// TwinCAT 3 PLC project Main
// ProgramVersion: 3.1.4026.10
// libraries:
//   Tc2_EtherCAT, * (Beckhoff Automation GmbH)
//   Tc2_IoFunctions, * (Beckhoff Automation GmbH)
//   Tc2_Math, * (Beckhoff Automation GmbH)
//   Tc2_MC2, * (Beckhoff Automation GmbH)
//   Tc2_NC, * (Beckhoff Automation GmbH)
//   Tc2_Standard, * (Beckhoff Automation GmbH)
//   Tc2_System, * (Beckhoff Automation GmbH)
//   Tc2_Utilities, * (Beckhoff Automation GmbH)
//   Tc3_EventLogger, * (Beckhoff Automation GmbH)
//   Tc3_McCollisionAvoidance, * (Beckhoff Automation GmbH)
//   Tc3_McCoordinatedMotion, * (Beckhoff Automation GmbH)
//   Tc3_Module, * (Beckhoff Automation GmbH)
//   Tc3_XTS_Utility, * (Beckhoff Automation GmbH)
// project tree:
//   DUTs/delete/ MainCommands_typ.TcDUT (not stored), MainStateMachine_enum.TcDUT, MainState_enum.TcDUT (not stored), MediatorGroupStatus.TcDUT (not stored), MotionParameters_typ.TcDUT (not stored), MoverCommandType_enum.TcDUT (not stored), MoverState_enum.TcDUT (not stored), PositionTriggerStats_typ.TcDUT (not stored), StationStats_typ.TcDUT (not stored), TrackCyclicState.TcDUT (not stored), TrackInfo.TcDUT (not stored), TrackState.TcDUT (not stored), UserStationsMonitor.TcDUT
//   DUTs/ M1Detection.TcDUT, MoverControlFlags.TcDUT, MoverSequence.TcDUT (not stored), StationSequence.TcDUT, XTSSequence.TcTLEO
//   / GlobalTextList.TcGTLO (not stored), PlcTask.TcTTO (not stored)
//   GVLs/ GVL.TcGVL, HMI.TcGVL, IOGVL.TcGVL, PersistentGVL.TcGVL, SafetyGVL.TcGVL
//   ITFs/ iMoverList.TcIO, iMover.TcIO (not stored), iTrack.TcIO
//   POUs/ Main.TcPOU
//   POUs/XTS/ Mover.TcPOU, Station.TcPOU

// ---- DUTs/delete/MainStateMachine_enum.TcDUT
{attribute 'strict'}
{attribute 'to_string'}
TYPE MainStateMachine_enum :
(
	MS_DISABLED			:= 0,
	MS_INITIALIZING		:= 10,
	MS_ENABLED			:= 20,
	MS_RUN				:= 30,
	MS_STOPPING			:= 40,
	MS_STOPPED			:= 50,
	MS_DISABLING		:= 60,
	MS_ERROR			:= 70,
	MS_DEBUG			:= 80	
);
END_TYPE

// ---- DUTs/delete/UserStationsMonitor.TcDUT
TYPE UserStationsMonitor :
STRUCT
	
bmoverAtStation		: ARRAY[0..GVL.NUM_STATIONS] OF BOOL;
nmoverAtStation		: ARRAY[0..GVL.NUM_STATIONS] OF UDINT;


END_STRUCT
END_TYPE

// ---- DUTs/M1Detection.TcDUT
{attribute 'qualified_only'}
{attribute 'strict'}
{attribute 'to_string'}
TYPE M1Detection :
(
	Read,
	ReadBuffer,
	Analyze,
	Write,
	WriteBuffer,
	Done,
	Error
	
);
END_TYPE

// ---- DUTs/MoverControlFlags.TcDUT
TYPE MoverControlFlags :
STRUCT

	loadTray_Busy		: BOOL;			// To the machine to check Sensor
	loadTray_Complete	: BOOL;			// From Sensor is TRUE
	inspectTray_Busy	: BOOL;			// Read the state of the sensor TRUE/FALSE
	inspectTray_Complate: BOOL;			// From Camera that tray is done being measured
	loadArea1_Busy		: BOOL;			// TO Robot 1 to start working
	loadArea1_Complete	: BOOL;			// FROM Robot 1 that placing parts has completed
	loadArea2_Busy		: BOOL;			// TO Robot 2 to start working
	loadArea2_Complete	: BOOL;			// FROM Robot 1 that placing parts has completed
	loadArea3_Busy		: BOOL;			// TO Robot 3 to start working
	loadArea3_Complete	: BOOL;			// FROM Robot 1 that placing parts has completed
	loadArea4_Busy		: BOOL;			// TO Robot 4 to start working
	loadArea4_Complete	: BOOL;			// From Robot 1 that placing parts has completed
	unloadTray_Busy		: BOOL;			// To Robot 5 to start working
	unloadTray_Complete	: BOOL;			// From Robot 5. Tray is unloaded



END_STRUCT
END_TYPE

// ---- DUTs/StationSequence.TcDUT
{attribute 'qualified_only'}
{attribute 'strict'}
TYPE StationSequence :
(
	Idle,
	MoverPresent,
	RobotActive,
	DischargeMover,
	Error		
);
END_TYPE

// ---- DUTs/XTSSequence.TcTLEO
{attribute 'qualified_only'}
{attribute 'strict'}
{attribute 'to_string'}
TYPE XTSSequence :
(
	Off,
	EnableMovers,
	EnableGroup,
	AddAxes,
	RemoveAxes,
	RemovedAxes,
	DisableMovers,
	Disabled,
	Start,
	Run,
	Stop,
	Stopping,
	Paused,
	Standby,
	Error,
	Waiting
);
END_TYPE

// ---- GVLs/GVL.TcGVL
{attribute 'qualified_only'}
VAR_GLOBAL CONSTANT
	pXtsProcessingUnit 			: OTCID	:= 16#01010020;	 
	TRACK_LENGTH 				: LREAL := 7000; // This should be set to the exact length [mm] of the track system
	NUM_MOVERS   				: USINT := 20;   // This should be set to the exact number of movers on the system
	
	// The following should be set to a value **equal to or greater than** the number of objectives needed
	NUM_POSITIONTRIGGERS		: USINT := 10;	// Position Triggers
	NUM_STATIONS				: USINT := 8;	// Stations
	NUM_ZONES					: USINT := 10;	// Zones

	// Station constants
	startStation				: USINT	:= 1;		// set this number to the index of the station all movers should start from
	stationTolerance			: LREAL	:= 1;		// set to number of millimeters tolerance for mover at station
	zeroSpeed					: LREAL	:= 10.0;	// tolerance for definition of not moving
END_VAR

VAR_GLOBAL
	Mover					: ARRAY[1..GVL.NUM_MOVERS] OF Mover;
	Station					: ARRAY[1..GVL.NUM_STATIONS] OF station;
	dsMoverControlFlags		: MoverControlFlags;
END_VAR

// ---- GVLs/HMI.TcGVL
{attribute 'qualified_only'}
VAR_GLOBAL
	Start					: BOOL;
	ReStart					: BOOL;
	Stop					: BOOL;
	Resume					: BOOL;
	ResetXTS_Error			: BOOL;
	dsMoverControlFlags		: MoverControlFlags;
	ShuttleMover			: BOOL;
	MachineState			: STRING;
	AutoMode				: BOOL;
	
	//Linked to SAFETY Alias
	LockDoors		AT %Q*	: BOOL;		
	
END_VAR

// ---- GVLs/IOGVL.TcGVL
{attribute 'qualified_only'}
VAR_GLOBAL
	
//INPUTS
iTrayDetectSensor	AT %I*	:	BOOL;
iDoor1Opened		AT %I*	:	BOOL;		
iDoor2Opened		AT %I*	:	BOOL;
iDoor3Opened		AT %I*	:	BOOL;
iDoor4Opened		AT %I*	:	BOOL;
iMainAirPressure 	AT %I*	:	BOOL;

//------XTS Power Monitor Breakers	
//- EL1809 Mod1
iCircuitBreaker24VDC			AT %I*	:	BOOL;
iCircuitBreakerSafety			AT %I*	:	BOOL;
iXTS_Module1					AT %I*	:	BOOL;
iXTS_Module2					AT %I*	:	BOOL;
iXTS_Module3					AT %I*	:	BOOL;
iXTS_Module4					AT %I*	:	BOOL;
iXTS_Module5					AT %I*	:	BOOL;
iXTS_Module6					AT %I*	:	BOOL;
iLubricationOn					AT %I*	:	BOOL;
//- EL1809 Mod2
iPowerSupply48VDC1				AT %I*	:	BOOL;
iPowerSupply48VDC2				AT %I*	:	BOOL;
iPowerSupply48VDC3				AT %I*	:	BOOL;
iLubricationLevelOK				AT %I*	:	BOOL;
iLubricationDone				AT %I*	:	BOOL;
iCircuitBreaker48VDC1			AT %I*	:	BOOL;
iCircuitBreaker48VDC2			AT %I*	:	BOOL;
iCircuitBreaker48VDC3			AT %I*	:	BOOL;
iCircuitBreakerXTSModule1		AT %I*	:	BOOL;
iCircuitBreakerXTSModule2		AT %I*	:	BOOL;
iCircuitBreakerXTSModule3		AT %I*	:	BOOL;
iCircuitBreakerXTSModule4		AT %I*	:	BOOL;
iCircuitBreakerXTSModule5		AT %I*	:	BOOL;
iCircuitBreakerXTSModule6		AT %I*	:	BOOL;
iBrakeResistorON				AT %I*	:	BOOL;

//-----------------------------------------------------------------------------------------------------------------------------------
//OUTPUTS
oBacklight1			AT %Q*	:	BOOL;
oBacklight2			AT %Q*	:	BOOL;
oBacklight3			AT %Q*	:	BOOL;
oBacklight4			AT %Q*	:	BOOL;
oBacklight5			AT %Q*	:	BOOL;
oBacklight6			AT %Q*	:	BOOL;
oBacklight7			AT %Q*	:	BOOL;
oBacklight8			AT %Q*	:	BOOL;
oBacklight9			AT %Q*	:	BOOL;
oBacklight10		AT %Q*	:	BOOL;
oBacklight11		AT %Q*	:	BOOL;
oBacklight12		AT %Q*	:	BOOL;
oBacklight13		AT %Q*	:	BOOL;
oBacklight14		AT %Q*	:	BOOL;
oBacklight15		AT %Q*	:	BOOL;
oBacklight16		AT %Q*	:	BOOL;
oEStopLight			AT %Q*	:	BOOL;
oConveyor			AT %Q*	:	BOOL;
oLubeON				AT %Q*	:	BOOL;

END_VAR

// ---- GVLs/PersistentGVL.TcGVL
{attribute 'qualified_only'}

VAR_GLOBAL RETAIN
	
TimesAroundTrackCounter		: INT;

END_VAR

// ---- GVLs/SafetyGVL.TcGVL
{attribute 'qualified_only'}
VAR_GLOBAL
	
//OUTPUTS TO SAFETY GROUP
err_ack			AT %Q*	:	BOOL;
run				AT %Q*	:	BOOL := TRUE;
DoorsClosed 	AT %Q*	:	BOOL;
ResetCurtains	AT %Q*	:	BOOL;

//INPUTS FROM SAFETY GROUP
CurtainsOK		AT %I*	:	BOOL;
AllSafetyOK		AT %I*	:	BOOL;
EStopStatus		AT %I*	:	BOOL;
DoorsLocked		AT %I*	:	BOOL;

END_VAR

// ---- ITFs/iMoverList.TcIO
INTERFACE iMoverList

METHOD ActivateAllTrack : BOOL
VAR_INPUT
	Track	: REFERENCE TO Track;
END_VAR
END_METHOD

METHOD ApplyAllParameterSet : iMoverList
VAR_INPUT
	ParameterSet		: MotionParameters_typ;
END_VAR
END_METHOD

METHOD Contains : BOOL
VAR_INPUT
	
	Mover		: REFERENCE TO delete_Mover;

END_VAR
END_METHOD

METHOD DestinationStation : iMoverList
VAR_INPUT
	Destination	: REFERENCE TO delete_Station;
END_VAR
END_METHOD

METHOD DisableAll : iMoverList
END_METHOD

METHOD EnableAll : iMoverList
END_METHOD

METHOD GetMoverByLocation : REFERENCE to delete_Mover
VAR_INPUT
    Index     : USINT;                // 0 is find the first closest mover, 1 is find the second closest mover, 2 is find the third, etc. etc. etc.
    Position  : LREAL;                // Fixed track position from which to search for movers by proximity
    Direction : Tc2_MC2.MC_Direction; // Positive = find the most positive mover whose position is less than the Input. Negative = find the most negative mover whose position is greater than the input
END_VAR
END_METHOD

METHOD HaltAll : iMoverList
END_METHOD

PROPERTY IsAllMoversDisabled : bool
GET
END_GET
END_PROPERTY

PROPERTY IsAllMoversHalted : bool
GET
END_GET
END_PROPERTY

PROPERTY IsAllMoversReady : BOOL
GET
END_GET
END_PROPERTY

PROPERTY IsAllTrackReady : BOOL
GET
END_GET
END_PROPERTY

METHOD LogicalComplement : MoverList
VAR_INPUT
END_VAR
END_METHOD

METHOD LogicalDifference : MoverList
VAR_INPUT
	
	MoverList		: MoverList;

END_VAR
END_METHOD

METHOD LogicalIntersect : MoverList
VAR_INPUT
	
	MoverList		: MoverList;

END_VAR
END_METHOD

METHOD LogicalUnion : MoverList
VAR_INPUT
	
	MoverList		: MoverList;

END_VAR
END_METHOD

METHOD MoveAllToPosition : iMoverList
VAR_INPUT

    DestinationPosition : LREAL; // position on track for all shuttles to move towards	

END_VAR
END_METHOD

METHOD MoveAllToStation : iMoverList
VAR_INPUT

    DestinationStation : REFERENCE TO delete_Station;

END_VAR
END_METHOD

METHOD MoveAllVelocity : iMoverList
VAR_INPUT

    Velocity : LREAL;

END_VAR
END_METHOD

METHOD SetAllAcceleration : iMoverList
VAR_INPUT

    Acceleration : LREAL;

END_VAR
END_METHOD

METHOD SetAllDeceleration : iMoverList
VAR_INPUT

    Deceleration : LREAL;

END_VAR
END_METHOD

METHOD SetAllDirection : iMoverList
VAR_INPUT

    Direction : Tc3_Mc3Definitions.MC_DIRECTION;

END_VAR
END_METHOD

METHOD SetAllGap : iMoverList
VAR_INPUT
	Gap : LREAL;
END_VAR
END_METHOD

METHOD SetAllGapMode : iMoverList
VAR_INPUT
    Mode	: MC_GAP_CONTROL_MODE;
END_VAR
END_METHOD

METHOD SetAllJerk : iMoverList
VAR_INPUT

    Jerk : LREAL;

END_VAR
END_METHOD

METHOD SetAllVelocity : iMoverList
VAR_INPUT

    Velocity : LREAL;

END_VAR
END_METHOD

{attribute 'monitoring' := 'call'}
PROPERTY TrackedMoverCount : USINT
GET
END_GET
END_PROPERTY

PROPERTY TrackedMovers : ARRAY[0..GVL.NUM_MOVERS - 1] OF POINTER TO delete_Mover
GET
END_GET
END_PROPERTY

METHOD UnregisterAll : BOOL
VAR_INPUT
END_VAR
END_METHOD

END_INTERFACE

// ---- ITFs/iTrack.TcIO
INTERFACE iTrack

PROPERTY CurrentMoverCount : DINT
GET
END_GET
END_PROPERTY

PROPERTY CurrentMoverList : iMoverList
GET
END_GET
END_PROPERTY

METHOD Cyclic : BOOL
VAR_INPUT
END_VAR
END_METHOD

PROPERTY Id : INT
GET
END_GET
SET
END_SET
END_PROPERTY

PROPERTY isInitialized : bool
GET
END_GET
END_PROPERTY

PROPERTY OTCID : OTCID
GET
END_GET
SET
END_SET
END_PROPERTY

METHOD RegisterMover : BOOL
VAR_INPUT
    NewMover : REFERENCE TO delete_Mover;
END_VAR
VAR
END_VAR
END_METHOD

METHOD UnregisterAll : BOOL
VAR_INPUT
END_VAR
END_METHOD

METHOD UnregisterMover : BOOL
VAR_INPUT
    RemovingMover : REFERENCE TO delete_Mover;
END_VAR
VAR
END_VAR
END_METHOD

END_INTERFACE

// ---- POUs/XTS/Station.TcPOU
FUNCTION_BLOCK Station
VAR_INPUT
	Position		: LREAL;
	bMoveToNext		: BOOL;
	bMoveToStart	: BOOL;
	bMoveToQueue	: BOOL;
END_VAR
VAR_OUTPUT
	CurrentMover	: UDINT;
END_VAR
VAR
	Step			: StationSequence;
	i				: USINT;
	PosLow			: LREAL;
	PosHigh			: LREAL;
END_VAR

(* this function block handles each station *)

PosLow		:= Position - ( GVL.stationTolerance / 2 );
IF PosLow < 0 THEN
	PosLow	:= GVL.TRACK_LENGTH + PosLow;
END_IF
PosHigh		:= Position + ( GVL.stationTolerance / 2 );


CASE Step OF 
//-----------------------------------------------------------------------------------------------------------------------	
	StationSequence.Idle:
		// loop through all movers checking position
		FOR i := 1 TO GVL.NUM_MOVERS DO
			IF GVL.Mover[i].Ready
			AND ( GVL.Mover[i].Step = MoverSequence.AtStart OR GVL.Mover[i].Step = MoverSequence.AtStation )
			AND ABS(GVL.Mover[i].Velocity) < GVL.zeroSpeed THEN
				IF PosLow < PosHigh THEN
					IF GVL.Mover[i].Position > PosLow
					AND GVL.Mover[i].Position < PosHigh THEN
						CurrentMover	:= i;
						Step			:= StationSequence.MoverPresent;
					END_IF
				ELSE
					// station position is close to rollover
					IF GVL.Mover[i].Position > PosLow
					OR GVL.Mover[i].Position < PosHigh THEN
						CurrentMover	:= i;
						Step			:= StationSequence.MoverPresent;
					END_IF
				END_IF
			END_IF
		END_FOR
		
//-----------------------------------------------------------------------------------------------------------------------	
	StationSequence.MoverPresent:
		// robot tasks complete, discharge mover
		IF bMoveToNext THEN									
			Step	:= StationSequence.Idle;
			bMoveToNext := FALSE;
			GVL.Mover[CurrentMover].toNext	:= TRUE;		// request mover move to next station
		END_IF
		
		IF bMoveToStart THEN
			Step	:= StationSequence.Idle;
			bMoveToStart := FALSE;
			GVL.Mover[CurrentMover].toStart	:= TRUE;		// request mover move to Start station
		END_IF
		
		IF bMoveToQueue THEN
			Step	:= StationSequence.Idle;
			bMoveToQueue := FALSE;
			GVL.Mover[CurrentMover].toQueue	:= TRUE;
		END_IF

		
//-----------------------------------------------------------------------------------------------------------------------		
	StationSequence.DischargeMover:
		// request mover move to next station
		//GVL.Mover[CurrentMover].toNext	:= TRUE;
		// verify mover has left
		IF GVL.Mover[CurrentMover].Busy
			AND GVL.Mover[CurrentMover].Position > (Position + GVL.stationTolerance / 2)
			AND GVL.Mover[CurrentMover].Velocity > GVL.zeroSpeed THEN
			Step	:= StationSequence.Idle;
		END_IF
		
END_CASE

END_FUNCTION_BLOCK

// ---- POUs/XTS/Mover.TcPOU
FUNCTION_BLOCK Mover
VAR_INPUT
	Enable			: BOOL;				// Request mover enable
	toStart			: BOOL;				// Request mover go to start position
	toNext			: BOOL;				// Request mover go to next station	
	toStop			: BOOL;				// Request mover to stop - meaning the movers will be stop, removed from group, and power will be shutdown to the track via an E-Stop or HMI.Stop	
	toPause			: BOOL;				// Request mover to pause	
	toDisable		: BOOL;				// Request mover to disable power	
	toQueue			: BOOL;				// Request current mover at starting station to join the back of the queue
	toReset			: BOOL;				// Request current mover at starting station to join the back of the queue
	toIncreaseSpeed	: BOOL;
END_VAR
VAR_OUTPUT
	Enabled			: BOOL;				// Mover confirmed enabled
	Ready			: BOOL;				// Mover is enabled and ready to accept motion commands
	Busy			: BOOL;				// Mover is processing a command or changing state
	Position		: LREAL;			// Current mover position
	Velocity		: LREAL;			// Current mover velocity                                	
	Error			: UDINT;			// errorID of the active error
	Step			: MoverSequence;	// Mover's step within sequence                                	
	AxisReference	: AXIS_REF;			// Motion link variable. Left as output so the link can be made directly, and accessed by external code
	TargetStation	: USINT;
END_VAR
VAR
	// Motion commands
	fbPower					: MC_Power;
	fbReset					: MC_Reset;
	fbHaltCA				: MC_HaltCA;
	fbMoveAbsCA				: MC_MoveAbsoluteCA;
	fbMoveAbsCABlended		: MC_MoveAbsoluteCA;
	fbMoveAbsCABlended2		: MC_MoveAbsoluteCA;
	
	MoveCommandVel			: LREAL := 1000;
	PosLow					: LREAL;
	PosHigh					: LREAL;
	bDummySpeedTest			: BOOL;
	
END_VAR

(* this function block handles each Mover's axis *)

	AxisReference.ReadStatus();
	Enabled		:= NOT AxisReference.Status.Disabled;
	Ready		:= AxisReference.Status.NotMoving AND NOT AxisReference.Status.Error AND NOT AxisReference.Status.Disabled;
	Busy		:= AxisReference.Status.Moving;
	Position	:= AxisReference.NcToPlc.ModuloActPos;
	Velocity	:= AxisReference.NcToPlc.ActVelo;
	Error		:= AxisReference.NcToPlc.ErrorCode;
	
	IF Step = MoverSequence.AtStart AND toQueue THEN
		Step := MoverSequence.MovingToQueue;
		toQueue := FALSE;
	END_IF
	
	IF toStop OR toPause THEN
		fbMoveAbsCA.Execute			:= FALSE;
		fbMoveAbsCABlended.Execute	:= FALSE;
		fbHaltCA.Execute 			:= TRUE;
		fbHaltCA.Deceleration 		:= 1E4;
		IF toStop THEN
			Step := MoverSequence.Stopping;
		ELSIF toPause THEN
			Step := MoverSequence.Pausing;
		END_IF
	END_IF
	
	IF toReset THEN
		Step := MoverSequence.Reset;
		toReset := FALSE;
	END_IF
	

CASE Step OF
//-----------------------------------------------------------------------------------------------------------------------
	MoverSequence.Reset:	
	
		fbReset.Execute := TRUE;
		IF fbReset.Busy THEN
			Step := MoverSequence.Resetting;
		END_IF
	
//---------------------------------
	MoverSequence.Resetting:	
	
	IF fbReset.Done THEN
		fbReset.Execute := FALSE;
		Step := MoverSequence.Waiting;
	END_IF

//-----------------------------------------------------------------------------------------------------------------------
	MoverSequence.MovingToQueue:	
	
		IF NOT fbMoveAbsCA.Busy AND NOT fbMoveAbsCA.Done THEN			//Add additional condition that the doors are not unlcoked
			fbMoveAbsCA.Execute			:= TRUE;
			fbMoveAbsCA.Position		:= GVL.Station[GVL.startStation].Position+2000;
			fbMoveAbsCA.Velocity		:= MoveCommandVel;										// parameterize
			fbMoveAbsCA.Direction		:= MC_Positive_Direction;						// usually positive
		END_IF
			// check for error
		IF fbMoveAbsCA.Error THEN
			Error				:= fbMoveAbsCA.ErrorId;
			Step				:= MoverSequence.Error;
			fbMoveAbsCA.Execute	:= FALSE;
		END_IF
		// check for move complete THEN proceed to starting station
		IF fbMoveAbsCA.Busy AND Position > 1500.0 AND Position < 6900.0 THEN 		//When mover sits at position 0 the values jump +-0 so an asdditional condition must be used
			fbMoveAbsCABlended.Execute		:= TRUE;
			fbMoveAbsCABlended.Position		:= GVL.Station[GVL.startStation].Position;
			fbMoveAbsCABlended.Velocity		:= MoveCommandVel;
			fbMoveAbsCABlended.BufferMode	:= mcAborting;
			fbMoveAbsCABlended.Direction 	:= MC_Positive_Direction;
			Step							:= MoverSequence.AtQueue;
		END_IF
		
//---------------------------------
	MoverSequence.AtQueue:	
	
		IF fbMoveAbsCABlended.Busy THEN
			fbMoveAbsCABlended.Execute			:= FALSE;
			fbMoveAbsCA.Execute					:= FALSE;
			Step								:= MoverSequence.MovingToStart;
		END_IF
	
//-----------------------------------------------------------------------------------------------------------------------
	MoverSequence.Stopping:	
		//RESULT OF PRESSING ESTOP
		IF fbHaltCA.Done OR AxisReference.Status.StandStill OR AxisReference.Status.NotMoving THEN
			fbHaltCA.Execute 	:= FALSE;
			toStart				:= FALSE;
			toNext				:= FALSE;
			toStop				:= FALSE;
			Step := MoverSequence.Disabling;
		END_IF
			
//---------------------------------
	MoverSequence.Disabling:		
	 	//RESULT OF PRESSING ESTOP
		IF toDisable THEN
			Enable						:= FALSE;
			fbPower.Enable				:= FALSE;
			fbPower.Enable_Positive		:= FALSE;
			fbPower.Enable_Negative		:= FALSE;
			fbPower.BufferMode			:= MC_Aborting;
			fbPower.Override			:= 100;
			IF AxisReference.Status.Disabled THEN
				toDisable := FALSE;
				Step := MoverSequence.Off;
			END_IF
		END_IF
			
//-----------------------------------------------------------------------------------------------------------------------
	MoverSequence.Pausing:	
	
		IF fbHaltCA.Done THEN
			fbHaltCA.Execute 	:= FALSE;
			toStart				:= FALSE;
			toNext				:= FALSE;
			toPause				:= FALSE;
			Step := MoverSequence.OFF;
		END_IF

//---------------------------------
	MoverSequence.Off:
		// when enable request is true, use MC_Power function block
		IF Enable THEN
			fbPower.Enable_Positive := TRUE;
			fbPower.Enable := TRUE;
		END_IF
		IF Enabled THEN
			Step	:= MoverSequence.Idle;
		END_IF
		
//---------------------------------	
	MoverSequence.Idle:
		// ready and awaiting either toStart or toNext
		IF toStart THEN
			TargetStation		:= GVL.startStation;
			Step				:= MoverSequence.MovingToStart;
		ELSIF toNext THEN
			Step				:= MoverSequence.MovingToStation;
		END_IF
		
//-----------------------------------------------------------------------------------------------------------------------	
	MoverSequence.MovingToStart:
		// move absolute with collision avoidance to start station
		IF NOT fbMoveAbsCA.Busy AND NOT fbMoveAbsCA.Done THEN	
			fbMoveAbsCA.Execute		:= TRUE;
			fbMoveAbsCA.Position	:= GVL.Station[GVL.startStation].Position;
			fbMoveAbsCA.Velocity	:= MoveCommandVel;							// parameterize
			fbMoveAbsCA.Direction	:= MC_Positive_Direction;		// usually positive
		END_IF
		// check for error
		IF fbMoveAbsCA.Error THEN
			Error				:= fbMoveAbsCA.ErrorId;
			Step				:= MoverSequence.Error;
			fbMoveAbsCA.Execute	:= FALSE;
		END_IF
		IF fbMoveAbsCA.Busy AND Position > GVL.Station[8].Position OR Position < GVL.Station[1].Position THEN
			fbMoveAbsCABlended.Execute		:= TRUE;
			fbMoveAbsCABlended.Position	:= GVL.Station[GVL.startStation].Position;
			fbMoveAbsCABlended.Velocity	:= 100;
			fbMoveAbsCABlended.BufferMode	:= mcAborting;
			fbMoveAbsCABlended.Direction 	:= MC_Positive_Direction;
			bDummySpeedTest := TRUE;
		END_IF
		// check for move complete
		IF fbMoveAbsCA.Done OR fbMoveAbsCABlended2.Done OR (Position > (GVL.Station[1].Position - 3) AND Position < (GVL.Station[1].Position + 3)) THEN
			fbMoveAbsCA.Execute			:= FALSE;
			fbMoveAbsCABlended.Execute	:= FALSE;
			toStart						:= FALSE;
			Step						:= MoverSequence.AtStart;
		END_IF
		
//-----------------------------------------------------------------------------------------------------------------------	
	MoverSequence.AtStart:
		toStart					:= FALSE;							//Add additional condition that the doors are not unlcoked
		// wait for command to next station
		IF toNext THEN
			IF TargetStation < GVL.NUM_STATIONS THEN
				// next station
				TargetStation	:= TargetStation + 1;
			ELSE
				// at last station, next station is 1
				TargetStation	:= 1;
			END_IF
			Step				:= MoverSequence.MovingToStation;
		END_IF
		
//-----------------------------------------------------------------------------------------------------------------------	
	MoverSequence.MovingToStation:
		// move absolute with collision avoidance to next station		//Add additional condition that the doors are not unlcoked
		fbMoveAbsCA.Execute		:= TRUE;
		fbMoveAbsCA.Position	:= GVL.Station[TargetStation].Position;
		fbMoveAbsCA.Velocity	:= 100;										// parameterize
		fbMoveAbsCA.Direction	:= MC_Positive_Direction;					// usually positive
		// check for error
		IF fbMoveAbsCA.Error THEN
			Error				:= fbMoveAbsCA.ErrorId;
			Step				:= MoverSequence.Error;
			fbMoveAbsCA.Execute	:= FALSE;
		END_IF
		IF fbMoveAbsCA.Busy AND Position > GVL.Station[1].Position + 250 AND Position < GVL.Station[8].Position THEN
			fbMoveAbsCABlended.Execute		:= TRUE;
			fbMoveAbsCABlended.Position		:= GVL.Station[TargetStation].Position;
			fbMoveAbsCABlended.Velocity		:= MoveCommandVel;
			fbMoveAbsCABlended.BufferMode	:= mcAborting;
			fbMoveAbsCABlended.Direction 	:= MC_Positive_Direction;
		END_IF
		// check for move complete
		IF fbMoveAbsCA.Done OR fbMoveAbsCABlended.Done THEN
			fbMoveAbsCA.Execute 		:= FALSE;
			fbMoveAbsCABlended.Execute	:= FALSE;
			toNext						:= FALSE;
			Step						:= MoverSequence.AtStation;
		END_IF
		
//-----------------------------------------------------------------------------------------------------------------------	
	MoverSequence.AtStation:
		// wait for command to next station
		IF toNext THEN															//Add additional condition that the doors are not unlcoked
			IF TargetStation < GVL.NUM_STATIONS THEN
				// next station
				TargetStation	:= TargetStation + 1;
			ELSE
				// at last station, next station is 1
				TargetStation	:= 1;
			END_IF
			Step				:= MoverSequence.MovingToStation;
		END_IF	
		IF toStart THEN
			Step				:= MoverSequence.MovingToStart;
			TargetStation		:= 1;
		END_IF
		
END_CASE

	fbPower				(Axis := AxisReference);
	fbReset				(Axis := AxisReference);
	fbHaltCA			(Axis := AxisReference);
	fbMoveAbsCA			(Axis := AxisReference);
	fbMoveAbsCABlended	(Axis := AxisReference);

END_FUNCTION_BLOCK

// ---- POUs/Main.TcPOU
PROGRAM Main
VAR
	PowerOn					: BOOL	:= TRUE;	// initialize on, turn false on second scan
	FirstRun				: BOOL	:= TRUE;		// initialize on, turn false when system has reached starting postion 
	i						: UINT;								// loop index variable
	Step					: XTSSequence;						// primary sequencer
	stCaGroupRef			: AXES_GROUP_REF;
	fbEnableGroup			: MC_GroupEnable;
	fbAddAxis				: ARRAY[1..GVL.NUM_MOVERS] OF MC_AddAxisToGroup;
	fbRemoveAxisFromGroup	: ARRAY[1..GVL.NUM_MOVERS] OF MC_RemoveAxisFromGroup;
	nAtStart				: UINT;
	nToStart				: UINT;
	allMoversHalted			: BOOL;	
	allMoversEnabled		: BOOL := FALSE;
	MoversReady				: BOOL;
	Started					: BOOL;		
	Resumed					: BOOL;
	ReStarted				: BOOL;
	bLightCurtainEntered	: R_TRIG;
	bLightCurtainExited		: F_TRIG;
	bEstopPressed			: F_TRIG;
	safeToOpenDoors			: BOOL;
	allMoversNotMoving		: BOOL;
	DelayMoversTimer		: TON;
	
	//Timers for generating a pulse
	PulseTON	: TON;
	PulseTOF	: TOF;
	OnDuration	: TIME := T#500MS;
	OFFDuration	: TIME := T#1000MS;
	bCycleBit	: BOOL;

	//M1 Detection
	fbReadM1DetectMode		: ADSREAD;
	fbReadM1DetectValid		: ADSREAD;
	fbReadM1DetectActive	: ADSREAD;
	fbWriteM1Detect			: ADSWRITE;
	fbDelayM1Timer			: TON;
	IsIdDetectionActive		: BOOL;			// M1 Detection currently underway
	Mover1Found				: BOOL;			// M1 Detection has completed
	Mover1Error				: BOOL;			// M1 Detection has Failed
	M1DetectStep			: M1Detection;	
	M1DetectAttemptCounter	: INT;
	
	bOperatorLoadingTrays	: BOOL;
	StopMoversLoopActive	: BOOL;
	Station2TON				: TON;
	Station3TON				: TON;
	Station4TON				: TON;
	Station5TON				: TON;
	Station6TON				: TON;
	Station7TON				: TON;
	
	bDummyBit				: BOOL;
	//Test					: FB_TcIoXtsEnvironment;
	delayOperatorDone		: BOOL;
	tonDelayOperatorDone	: TON;
END_VAR

(* this program handles the main sequencer of this machine *)
//Machine State is used to display state to HMI
HMI.MachineState := TO_STRING(Step); 
//Test.XpuTcIo(1).MoverTcIo(1).GetDistanceDriven();

// cyclic call to execute fb's for movers
FOR i := 1 TO GVL.NUM_MOVERS DO
	GVL.Mover[i]();
	GVL.Mover[i].AxisReference.ReadStatus();
	fbRemoveAxisFromGroup[i](AxesGroup		:= stCaGroupRef);
	fbAddAxis[i](AxesGroup		:= stCaGroupRef,
				Axis			:= GVL.Mover[i].AxisReference);
	//Monitoring if all movers are in stopped motion state			
	IF GVL.Mover[i].AxisReference.Status.Moving THEN
		allMoversNotMoving	:= FALSE;
	ELSE
		allMoversNotMoving	:= TRUE;
	END_IF
END_FOR

// cyclic call to execute fb's for stations
FOR i := 1 TO GVL.NUM_STATIONS DO
	GVL.Station[i]();
END_FOR

IF HMI.ResetXTS_Error THEN
	FOR i := 1 TO GVL.NUM_MOVERS DO
		GVL.Mover[i].toReset := TRUE;
	END_FOR
	HMI.ResetXTS_Error := FALSE;
END_IF

// E_Stop will halt, disable, and remove power from track and movers
bEstopPressed(CLK:=SafetyGVL.EStopStatus);
IF bEstopPressed.Q THEN
	Step			:= XTSSequence.Stop;
END_IF

// HMI Stop creates a paused state
IF HMI.Stop THEN 
	Step			:= XTSSequence.Paused;
	HMI.Stop		:= FALSE;
END_IF

CASE Step OF
//-----------------------------------------------------------------------------------------------------------------------	
	XTSSequence.Off:
		IF SafetyGVL.EStopStatus AND IOGVL.iPowerSupply48VDC1 AND IOGVL.iPowerSupply48VDC2 AND IOGVL.iPowerSupply48VDC3 AND Mover1Found = FALSE THEN
			Initialize();
		END_IF
		// state waiting for HMI.Start
		IF HMI.Start AND Mover1Found THEN
			Step		:= XTSSequence.EnableMovers;
			Started 	:= TRUE;
			HMI.Start 	:= FALSE;
		END_IF

//-----------------------------------------------------------------------------------------------------------------------	
	XTSSequence.Paused:
	
	Station2TON.IN := FALSE;
	Station3TON.IN := FALSE;
	Station4TON.IN := FALSE;
	Station5TON.IN := FALSE;
	Station6TON.IN := FALSE;
	Station7TON.IN := FALSE;
	tonDelayOperatorDone.IN := FALSE;
	
	//state waiting for HMI.Start or HMI.Resume
	IF allMoversNotMoving AND SafetyGVL.AllSafetyOK AND bOperatorLoadingTrays = FALSE THEN	
		IF HMI.ReStart THEN
			ReStarted 	:= TRUE;
			HMI.ReStart := FALSE;
			HMI.Stop  	:= FALSE;
			Step		:= XTSSequence.EnableMovers;
		END_IF
	
		IF HMI.Resume THEN
			Step		:= XTSSequence.EnableMovers;
			Resumed 	:= TRUE;
			HMI.Resume 	:= FALSE;
			HMI.Stop  	:= FALSE;
		END_IF
	END_IF
			
//-----------------------------------------------------------------------------------------------------------------------	
	XTSSequence.Stop:
	
		FOR i := 1 TO GVL.NUM_MOVERS  DO
			GVL.Mover[i].toStop := TRUE;
		END_FOR
		
		Started 	:= FALSE;
		Resumed 	:= FALSE;
		Step		:= XTSSequence.Stopping;
		
//-----------------------------------------------------------------------------------------------------------------------	
	XTSSequence.Stopping:
		// Waiting for all to come to a full stop
		allMoversHalted		:= TRUE;
		
		FOR i := 1 TO GVL.NUM_MOVERS DO
			IF GVL.Mover[i].AxisReference.Status.Moving THEN
				allMoversHalted		:= FALSE;
			END_IF
		END_FOR
		
		IF allMoversHalted THEN
			Step := XTSSequence.RemoveAxes;
		END_IF
	
//-----------------------------------------------------------------------------------------------------------------------	
	XTSSequence.RemoveAxes:
		// remove all axes to collision avoidance group loop through each mover axis and remove CA group
		FOR i:= 1 TO GVL.NUM_MOVERS DO
			fbRemoveAxisFromGroup[i].IdentInGroup := UDINT_TO_IDENTINGROUP(UINT_TO_UDINT(i));
			fbRemoveAxisFromGroup[i].Execute			:= TRUE;
		END_FOR
	
		IF stCaGroupRef.NcToPlc.CA.Common.GroupAxesCount = 0 THEN
			FOR i:= 1 TO GVL.NUM_MOVERS DO
				fbRemoveAxisFromGroup[i].IdentInGroup	:= UDINT_TO_IDENTINGROUP(UINT_TO_UDINT(i));
				fbRemoveAxisFromGroup[i].Execute			:= FALSE;
				MoversReady := FALSE;
		END_FOR
			Mover1Found := FALSE;
			Step := XTSSequence.DisableMovers;
		END_IF

//-----------------------------------------------------------------------------------------------------------------------	
	XTSSequence.DisableMovers:
	
		FOR i := 1 TO GVL.NUM_MOVERS  DO
			GVL.Mover[i].toDisable := TRUE;
		END_FOR
		allMoversEnabled := FALSE;
		
		//Disabling Movers if there is E-Stop Condition. This requires all stations to reset themselves.
		Step := XTSSequence.Off;
		
//-----------------------------------------------------------------------------------------------------------------------			
	XTSSequence.EnableMovers:
		// enable all movers
		FOR i := 1 TO GVL.NUM_MOVERS DO
			IF NOT GVL.Mover[i].Enabled THEN
				GVL.Mover[i].Enable	:= TRUE;
			END_IF
		END_FOR
		
		// check for all enabled
		FOR i := 1 TO GVL.NUM_MOVERS DO
			IF NOT GVL.Mover[i].Enabled THEN
				// not enabled, leave for loop
				EXIT;
			END_IF
			// made it this far, all movers are enabled
			IF i = gvl.NUM_MOVERS THEN
				Step	:= XTSSequence.EnableGroup;
			END_IF
		END_FOR
		
//-----------------------------------------------------------------------------------------------------------------------		
	XTSSequence.EnableGroup:
		// enable CA group
		fbEnableGroup.Execute := TRUE;
		// verify group enabled successfully
		IF fbEnableGroup.Done = TRUE THEN
			fbEnableGroup.Execute := FALSE;
			Step := XTSSequence.AddAxes;
		END_IF
		
//-----------------------------------------------------------------------------------------------------------------------		
	XTSSequence.AddAxes:
		// add all axes to collision avoidance group
		// loop through each mover axis and add to CA group
		FOR i:= 1 TO GVL.NUM_MOVERS DO
			fbAddAxis[i].IdentInGroup := UDINT_TO_IDENTINGROUP(UINT_TO_UDINT(i));
			fbAddAxis[i].Execute := TRUE;
		END_FOR
		
		// verify all axes added
		IF stCaGroupRef.NcToPlc.CA.Common.GroupAxesCount = GVL.NUM_MOVERS THEN
			FOR i:= 1 TO GVL.NUM_MOVERS DO
				fbAddAxis[i].IdentInGroup := UDINT_TO_IDENTINGROUP(UINT_TO_UDINT(i));
				fbAddAxis[i].Execute := FALSE;
				Step	:= XTSSequence.StandBy;
				allMoversEnabled := TRUE;
			END_FOR
		END_IF
		
//-----------------------------------------------------------------------------------------------------------------------		
	XTSSequence.StandBy:
		IF Started OR Restarted THEN
			Started		:= FALSE;
			Restarted	:= FALSE;
			Step		:= XTSSequence.Start;
		ELSIF Resumed THEN
			Resumed := FALSE;
			Step	:= XTSSequence.Run;
		END_IF
		
//-----------------------------------------------------------------------------------------------------------------------		
	XTSSequence.Start:
		// request all movers proceed to starting station
		IF bOperatorLoadingTrays = FALSE THEN
			FOR i:= 1 TO GVL.NUM_MOVERS DO
				GVL.Mover[i].toStart	:= TRUE;
			END_FOR
			FOR i:= 2 TO GVL.NUM_STATIONS DO
				IF GVL.Station[i].Step = StationSequence.MoverPresent THEN
					GVL.Station[i].bMoveToStart	:= TRUE;
				END_IF
			END_FOR 
			Step	:= XTSSequence.Run;
		END_IF	
	
//-----------------------------------------------------------------------------------------------------------------------	
	XTSSequence.Run:
		// LOAD TRAY STATION
		IF GVL.Station[1].Step = StationSequence.MoverPresent THEN
			HMI.dsMoverControlFlags.loadTray_Busy := TRUE;
			IF HMI.AutoMode AND IOGVL.iTrayDetectSensor AND bOperatorLoadingTrays = FALSE  THEN			//IF SENSOR IS TRUE PACKAGE IS PRESENT MOVER GOES TO NEXT STATION
				IF delayOperatorDone = FALSE THEN
					GVL.Station[1].bMoveToNext := TRUE;
				END_IF
			ELSIF HMI.AutoMode AND IOGVL.iTrayDetectSensor AND bOperatorLoadingTrays THEN
				delayOperatorDone := TRUE;
			ELSIF HMI.dsMoverControlFlags.loadTray_Complete AND bOperatorLoadingTrays = FALSE THEN	
				HMI.dsMoverControlFlags.loadTray_Complete := FALSE;
				GVL.Station[1].bMoveToNext := TRUE;
			END_IF
		ELSE
			HMI.dsMoverControlFlags.loadTray_Busy := FALSE;
		END_IF
		
		IF delayOperatorDone AND bOperatorLoadingTrays = FALSE AND tonDelayOperatorDone.IN = FALSE THEN
			tonDelayOperatorDone(IN := TRUE, PT := T#1S);
		ELSIF tonDelayOperatorDone.Q THEN
			tonDelayOperatorDone.IN := FALSE;
			delayOperatorDone		:= FALSE;
		END_IF
		
//--------------------		
		// INSPECT TRAY STATION
		IF GVL.Station[2].Step = StationSequence.MoverPresent THEN
			HMI.dsMoverControlFlags.inspectTray_Busy := TRUE;			//Tell Robot Tray is present meaning this station is busy
			IF HMI.AutoMode THEN
 				IF Station2TON.IN = FALSE THEN
					Station2TON(IN := TRUE, PT := T#1S);
				END_IF
			ELSIF HMI.dsMoverControlFlags.inspectTray_Complate THEN
				HMI.dsMoverControlFlags.inspectTray_Complate := FALSE;
				GVL.Station[2].bMoveToNext := TRUE;
			END_IF
			IF Station2TON.Q AND GVL.Station[2].bMoveToNext = FALSE THEN
				Station2TON.IN := FALSE;
				GVL.Station[2].bMoveToNext := TRUE;
			END_IF
		ELSE
			HMI.dsMoverControlFlags.inspectTray_Busy := FALSE;
			Station2TON.IN := FALSE;
		END_IF
		
//--------------------		
		// LOAD PARTS STATION 1
		IF GVL.Station[3].Step = StationSequence.MoverPresent THEN
			HMI.dsMoverControlFlags.loadArea1_Busy := TRUE;			
			IF HMI.AutoMode THEN
 				IF Station3TON.IN = FALSE THEN
					Station3TON(IN := TRUE, PT := T#5S);
				END_IF
			ELSIF HMI.dsMoverControlFlags.loadArea1_Complete THEN
				HMI.dsMoverControlFlags.loadArea1_Complete := FALSE;
				GVL.Station[3].bMoveToNext := TRUE;
			END_IF
			IF Station3TON.Q AND GVL.Station[3].bMoveToNext = FALSE THEN
				Station3TON.IN := FALSE;
				GVL.Station[3].bMoveToNext := TRUE;
			END_IF
		ELSE
			HMI.dsMoverControlFlags.loadArea1_Busy := FALSE;
			Station3TON.IN := FALSE;
		END_IF
		
//--------------------			
		// LOAD PARTS STATION 2
		IF GVL.Station[4].Step = StationSequence.MoverPresent THEN
			HMI.dsMoverControlFlags.loadArea2_Busy := TRUE;			//Tell Robot Tray is present meaning this station is busy
			IF HMI.AutoMode THEN
 				IF Station4TON.IN = FALSE THEN
					Station4TON(IN := TRUE, PT := T#5S);
				END_IF
			ELSIF HMI.dsMoverControlFlags.loadArea2_Complete THEN
				HMI.dsMoverControlFlags.loadArea2_Complete := FALSE;
				GVL.Station[4].bMoveToNext := TRUE;
			END_IF
			IF Station4TON.Q AND GVL.Station[4].bMoveToNext = FALSE THEN
				Station4TON.IN := FALSE;
				GVL.Station[4].bMoveToNext := TRUE;
			END_IF
		ELSE
			HMI.dsMoverControlFlags.loadArea2_Busy := FALSE;
			Station4TON.IN := FALSE;
		END_IF
		
//--------------------		
		// LOAD PARTS STATION 3
		IF GVL.Station[5].Step = StationSequence.MoverPresent THEN
			HMI.dsMoverControlFlags.loadArea3_Busy := TRUE;			//Tell Robot Tray is present meaning this station is busy
			IF HMI.AutoMode THEN
 				IF Station5TON.IN = FALSE THEN
					Station5TON(IN := TRUE, PT := T#5S);
				END_IF
			ELSIF HMI.dsMoverControlFlags.loadArea3_Complete THEN
				HMI.dsMoverControlFlags.loadArea3_Complete := FALSE;
				GVL.Station[5].bMoveToNext := TRUE;
			END_IF
			IF Station5TON.Q AND GVL.Station[5].bMoveToNext = FALSE THEN
				Station5TON.IN := FALSE;
				GVL.Station[5].bMoveToNext := TRUE;
			END_IF
		ELSE
			HMI.dsMoverControlFlags.loadArea3_Busy := FALSE;
			Station5TON.IN := FALSE;
		END_IF
		
 //--------------------   	
		// LOAD PARTS STATION 4
		IF GVL.Station[6].Step = StationSequence.MoverPresent THEN
			HMI.dsMoverControlFlags.loadArea4_Busy := TRUE;			//Tell Robot Tray is present meaning this station is busy
			IF HMI.AutoMode THEN
 				IF Station6TON.IN = FALSE THEN
					Station6TON(IN := TRUE, PT := T#5S);
				END_IF
			ELSIF HMI.dsMoverControlFlags.loadArea4_Complete THEN
				HMI.dsMoverControlFlags.loadArea4_Complete := FALSE;
				GVL.Station[6].bMoveToNext := TRUE;
			END_IF
			IF Station6TON.Q AND GVL.Station[6].bMoveToNext = FALSE THEN
				Station6TON.IN := FALSE;
				GVL.Station[6].bMoveToNext := TRUE;
			END_IF
		ELSE
			HMI.dsMoverControlFlags.loadArea4_Busy := FALSE;
			Station6TON.IN := FALSE;
		END_IF
		
//--------------------
// UNLOAD PARTS STATION 
		IF GVL.Station[7].Step = StationSequence.MoverPresent THEN
			HMI.dsMoverControlFlags.unloadTray_Busy := TRUE;			//Tell Robot Tray is present meaning this station is busy
			IF HMI.AutoMode THEN
 				IF Station7TON.IN = FALSE THEN
					Station7TON(IN := TRUE, PT := T#4S);
				END_IF
			ELSIF HMI.dsMoverControlFlags.unloadTray_Complete THEN
				HMI.dsMoverControlFlags.unloadTray_Complete := FALSE;
				IF bOperatorLoadingTrays THEN
					GVL.Station[7].bMoveToNext := TRUE;					//Send to Queue Movers Station
				ELSE
					GVL.Station[7].bMoveToStart := TRUE;				//Send to Load Tray Station
				END_IF
			END_IF
			IF Station7TON.Q AND GVL.Station[7].bMoveToNext = FALSE THEN
				Station7TON.IN := FALSE;
				IF bOperatorLoadingTrays THEN
					GVL.Station[7].bMoveToNext := TRUE;					//Send to Queue Movers Station
				ELSE
					GVL.Station[7].bMoveToStart := TRUE;				//Send to Load Tray Station
				END_IF
			END_IF
		ELSE
			HMI.dsMoverControlFlags.unloadTray_Busy := FALSE;
			Station7TON.IN := FALSE;
		END_IF
		
//--------------------		
	// Queue Station used only if Operator is in Zone 1
		IF GVL.Station[8].Step = StationSequence.MoverPresent THEN
			IF bOperatorLoadingTrays = FALSE THEN			
				GVL.Station[8].bMoveToStart := TRUE;
			END_IF
		END_IF
		
END_CASE

fbEnableGroup(AxesGroup	:= stCaGroupRef);
LightCurtainCheck();
ShuttleMoverToQueue();
DoorsClosedMonitor();
Station2TON();
Station3TON();
Station4TON();
Station5TON();
Station6TON();
Station7TON();
tonDelayOperatorDone();

ACTION DoorsClosedMonitor:





IF IOGVL.iDoor1Opened OR IOGVL.iDoor2Opened OR IOGVL.iDoor3Opened OR IOGVL.iDoor4Opened THEN
	SafetyGVL.DoorsClosed := FALSE;
ELSE
	SafetyGVL.DoorsClosed := TRUE;
END_IF


PulseTON(IN := NOT SafetyGVL.AllSafetyOK AND NOT bCycleBit, PT := OnDuration);
PulseTOF(IN := bCycleBit, PT := OFFDuration);

IF PulseTON.Q THEN
	bCycleBit := TRUE;
	IOGVL.oEStopLight := TRUE;
ELSE 
	IOGVL.oEStopLight := FALSE;
END_IF

IF PulseTOF.Q THEN
	bCycleBit := FALSE;
END_IF
END_ACTION

METHOD Initialize : BOOL
VAR_INPUT
END_VAR
// set values of function blocks
	GVL.Station[1].Position		:= 15.67;				//	Load Tray
	GVL.Station[2].Position		:= 751.07;			//	Inspect Tray
	GVL.Station[3].Position		:= 1573.61;			//	Load Parts 1
	GVL.Station[4].Position		:= 2195.49;			//	Load Parts 2
	GVL.Station[5].Position		:= 2811.86;			//	Load Parts 3
	GVL.Station[6].Position		:= 3434.98;			//	Load Parts 4
	GVL.Station[7].Position		:= 4253.05;			//	Unload Tray
	GVL.Station[8].Position		:= 4667.05;			//	Queue Area if operator is in workspace
	
	CASE M1DetectStep OF		//This Case statement will make 10 attempts to find Mover1 and error if not successful
		
M1Detection.Read:// ------------------------------------------------------- Determine current M1 Detection Status
		
	fbWriteM1Detect.WRITE			:= FALSE;
	
	fbReadM1DetectValid.NETID		:= '';
	fbReadM1DetectValid.PORT		:= 351;
	fbReadM1DetectValid.IDXGRP		:= GVL.pXtsProcessingUnit;
	fbReadM1DetectValid.IDXOFFS		:= 16#03080251;
	fbReadM1DetectValid.LEN			:= SIZEOF( Mover1Found );
	fbReadM1DetectValid.DESTADDR	:= ADR( Mover1Found );
	fbReadM1DetectValid.READ		:= TRUE;
	
	fbReadM1DetectActive.NETID		:= '';
	fbReadM1DetectActive.PORT		:= 351;
	fbReadM1DetectActive.IDXGRP		:= GVL.pXtsProcessingUnit;
	fbReadM1DetectActive.IDXOFFS	:= 16#03080268;
	fbReadM1DetectActive.LEN		:= SIZEOF( IsIdDetectionActive );
	fbReadM1DetectActive.DESTADDR	:= ADR( IsIdDetectionActive );
	fbReadM1DetectActive.READ		:= TRUE;
	
	M1DetectStep 					:= M1Detection.ReadBuffer;
		
M1Detection.ReadBuffer:// ------------------------------------------------------- Buffer

	fbDelayM1Timer( IN := TRUE, PT := T#3000MS );
	IF fbDelayM1Timer.Q THEN
		fbDelayM1Timer.IN				:= FALSE;
		fbReadM1DetectValid.READ		:= FALSE;
		fbReadM1DetectActive.READ		:= FALSE;
		M1DetectAttemptCounter := M1DetectAttemptCounter + 1;
		M1DetectStep 			:= M1Detection.Analyze;
	END_IF
		
M1Detection.Analyze:// ------------------------------------------------------- Determine to activate M1 Detect or ignore
	
IF M1DetectAttemptCounter < 10 THEN
	IF IsIdDetectionActive THEN
		M1DetectStep					:= M1Detection.Read;
	ELSIF Mover1Found THEN
		M1DetectStep					:= M1Detection.Done;	// M1 Detection complete, ready to enable this mover
	ELSE
		M1DetectStep					:= M1Detection.Write;	// M1 Detection hasn't been started yet. So start it!	
	END_IF
ELSE
	M1DetectStep				:= M1Detection.Error;	// M1 Detection Failed
END_IF

M1Detection.Write:// ------------------------------------------------------- Begin M1 Detection

	fbWriteM1Detect.NETID			:= '';
	fbWriteM1Detect.PORT			:= 351;
	fbWriteM1Detect.IDXGRP			:= GVL.pXtsProcessingUnit;
	fbWriteM1Detect.IDXOFFS			:= 16#03080250;
	fbWriteM1Detect.WRITE			:= TRUE;

	M1DetectStep 					:= M1Detection.WriteBuffer;
		
M1Detection.WriteBuffer:// ------------------------------------------------------- Buffer

	fbDelayM1Timer( IN := TRUE, PT := T#2000MS );
		
	IF fbDelayM1Timer.Q THEN
		fbDelayM1Timer.IN				:= FALSE;
		fbWriteM1Detect.WRITE			:= FALSE;
		M1DetectStep 					:= M1Detection.Read;
	END_IF

M1Detection.Done:// ------------------------------------------------------- Finished M1 Detection

	Mover1Found := TRUE;
	IsIdDetectionActive := FALSE;
	M1DetectStep 					:= M1Detection.Read;

M1Detection.Error:// ------------------------------------------------------- Failed M1 Detection

	Mover1Error			:= TRUE;
	IsIdDetectionActive := FALSE;

END_CASE

fbReadM1DetectValid();
fbReadM1DetectActive();
fbWriteM1Detect();
fbDelayM1Timer();
END_METHOD

ACTION LightCurtainCheck:
// ZONE 0  OPERATER LOADING

IF SafetyGVL.CurtainsOK THEN
	bOperatorLoadingTrays := FALSE;
ELSE
	bOperatorLoadingTrays := TRUE;
END_IF


IF SafetyGVL.AllSafetyOK AND allMoversEnabled AND bOperatorLoadingTrays THEN

	FOR i:= 1 TO GVL.NUM_MOVERS DO	
		IF GVL.Mover[i].Position > 4500.0 OR GVL.Mover[i].Position < 250.0 THEN
			GVL.Mover[i].toPause	:= TRUE;
			GVL.Mover[i].toNext		:= FALSE;
			GVL.Mover[i].toStart	:= FALSE;
		END_IF
		DelayMoversTimer.IN := FALSE;
		StopMoversLoopActive := TRUE;
	END_FOR
	
END_IF	
	
IF bOperatorLoadingTrays = FALSE AND DelayMoversTimer.IN = FALSE AND StopMoversLoopActive THEN
	DelayMoversTimer( IN := TRUE, PT := T#1S );
	StopMoversLoopActive := FALSE;
END_IF
		
IF DelayMoversTimer.Q THEN
	FOR i:= 1 TO GVL.NUM_MOVERS DO	
		IF GVL.Mover[i].Position > 4500.0 OR GVL.Mover[i].Position < (GVL.Station[1].Position) THEN
			GVL.Mover[i].toStart	:= TRUE;
		ELSIF GVL.Mover[i].Position > (GVL.Station[1].Position + 1) AND GVL.Mover[i].Position < (GVL.Station[1].Position + 250) THEN
			GVL.Mover[i].toNext	:= TRUE;
		END_IF
	END_FOR
	DelayMoversTimer.IN := FALSE;
END_IF
    
DelayMoversTimer();
END_ACTION

ACTION ShuttleMoverToQueue:

// This will be used for set up if mover is needed to be re-circulated around track

IF 	GVL.Station[1].Step = StationSequence.MoverPresent AND 
	GVL.Station[2].Step = StationSequence.Idle AND 
	GVL.Station[3].Step = StationSequence.Idle AND 
	GVL.Station[4].Step = StationSequence.Idle AND 
	GVL.Station[5].Step = StationSequence.Idle AND 
	GVL.Station[6].Step = StationSequence.Idle AND 
	GVL.Station[7].Step = StationSequence.Idle AND 
	HMI.ShuttleMover THEN
		GVL.Station[1].bMoveToQueue := TRUE;
		HMI.ShuttleMover := FALSE;
END_IF
END_ACTION

END_PROGRAM
